(* CODESYS project EST_MULT.project

Project tree, tasks and I/O mapping:
  Device : CODESYS Control Win V3, 3S - Smart Software Solutions GmbH, order no. 305021, version 3.5.11.30
    application Application
      libraries: Standard, * (System)
      task MainTask (cyclic, interval t#20ms, priority 1) calls PLC_PRG
      program PLC_PRG [LD]
*)

// Device/Application/PLC_PRG
PROGRAM PLC_PRG
VAR
	S1 : BOOL;     // PARTE SISTEMA
    S2 : BOOL;     // PARA TUDO
    M2 : BOOL;     // ESTEIRA 2
    M1 : BOOL;     // ESTEIRA 1
    B1 : BOOL;     // FOTOCELULA SENSOR QUE DETECTA GARRAFAS PARA CONTAR
	P1: BOOL;
	P2: BOOL;
	P3: BOOL;
	P4: BOOL;
	CTU_1: CTU;
	CV1: WORD;
	TOF_1: TOF;
	ET1: TIME;
	P5: BOOL;
	AUX1: BOOL;
	ZERA : BOOL;
END_VAR
VAR // added by the converter: edge detectors and wires of the graphical bodies
    _ft1 : F_TRIG;
END_VAR

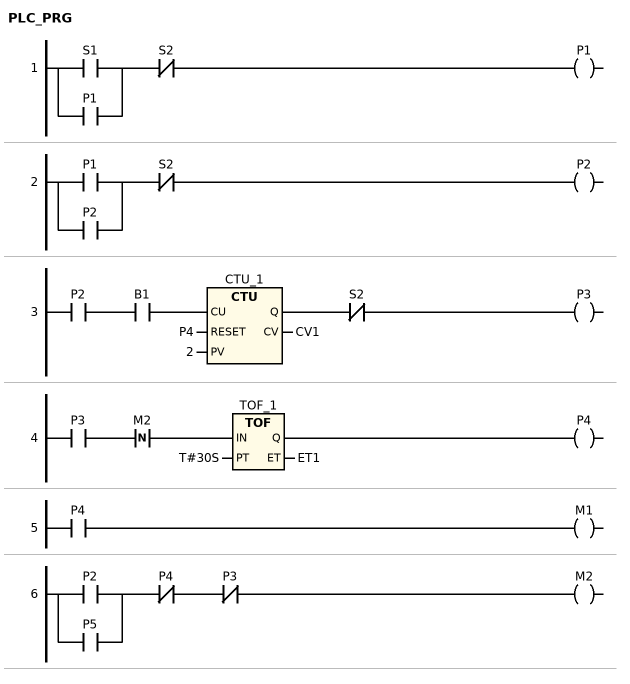
// NETWORK 1
P1 := (S1 OR P1) AND NOT S2;

// NETWORK 2
P2 := (P1 OR P2) AND NOT S2;

// NETWORK 3
CTU_1(CU := P2 AND B1, RESET := P4, PV := 2, CV => CV1); // CTU
P3 := CTU_1.Q AND NOT S2;

// NETWORK 4
_ft1(CLK := M2);
TOF_1(IN := P3 AND _ft1.Q, PT := T#30S, ET => ET1); // TOF
P4 := TOF_1.Q;

// NETWORK 5
M1 := P4;

// NETWORK 6
M2 := (P2 OR P5) AND NOT P4 AND NOT P3;

END_PROGRAM
